// TIA Portal V16 export
// export: Created 2022-11-01T21:54:10.5360386Z, ExportSetting WithDefaults, DisplayName Totally Integrated Automation Portal, DisplayVersion V16, DisplayName TIA Portal Version Control Interface, DisplayVersion V16, DisplayName TIA Portal Openness, DisplayVersion V16, DisplayName SINAMICS Startdrive Advanced, DisplayVersion V16, DisplayName SINAMICS Startdrive G130, G150, S120, S150, SINAMICS MV, S210, DisplayVersion V16, DisplayName SINAMICS Startdrive G110M, G120, G120C, G120D, G120P, DisplayVersion V16, DisplayName STEP 7 Professional, DisplayVersion V16, DisplayName STEP 7 Safety, DisplayVersion V16, DisplayName WinCC Professional, DisplayVersion V16
VAR_GLOBAL   // PLC tag table "DI/O C900"
   iH120_Run_Km AT %M2900.0 : Bool;
   iH120_Con_Vfd AT %M2900.1 : Bool;
   iH120_Run_Vfd AT %M2900.2 : Bool;
   "qH120_Sel_Loc/Rem" AT %M2900.3 : Bool;
   "qH120_Sel_Km/Vfd" AT %M2900.4 : Bool;
   qH120_Block AT %M2900.5 : Bool;
   qH120_Connect_Vfd AT %M2900.6 : Bool;
   qH120_Start AT %M2900.7 : Bool;
   "iH615/1_Run_Km" AT %M2901.0 : Bool;
   "iH615/1_Con_Vfd" AT %M2901.1 : Bool;
   "iH615/1_Run_Vfd" AT %M2901.2 : Bool;
   "qH615/1_Sel_Loc/Rem" AT %M2901.3 : Bool;
   "qH615/1_Sel_Km/Vfd" AT %M2901.4 : Bool;
   "qH615/1_Block" AT %M2901.5 : Bool;
   "qH615/1_Connect_Vfd" AT %M2901.6 : Bool;
   "qH615/1_Start" AT %M2901.7 : Bool;
   "iH615/2_Run_Km" AT %M2902.0 : Bool;
   "iH615/2_Con_Vfd" AT %M2902.1 : Bool;
   "iH615/2_Run_Vfd" AT %M2902.2 : Bool;
   "qH615/2_Sel_Loc/Rem" AT %M2902.3 : Bool;
   "qH615/2_Sel_Km/Vfd" AT %M2902.4 : Bool;
   "qH615/2_Block" AT %M2902.5 : Bool;
   "qH615/2_Connect_Vfd" AT %M2902.6 : Bool;
   "qH615/2_Start" AT %M2902.7 : Bool;
   "iH616-x/1_Run_Km" AT %M2903.0 : Bool;
   "iH616-x/1_Con_Vfd" AT %M2903.1 : Bool;
   "iH616-x/1_Run_Vfd" AT %M2903.2 : Bool;
   "qH616-x/1_Sel_Loc/Rem" AT %M2903.3 : Bool;
   "qH616-x/1_Sel_Km/Vfd" AT %M2903.4 : Bool;
   "qH616-x/1_Block" AT %M2903.5 : Bool;
   "qH616-x/1_Connect_Vfd" AT %M2903.6 : Bool;
   "qH616-x/1_Start" AT %M2903.7 : Bool;
   "iH616-x/2_Run_Km" AT %M2904.0 : Bool;
   "iH616-x/2_Con_Vfd" AT %M2904.1 : Bool;
   "iH616-x/2_Run_Vfd" AT %M2904.2 : Bool;
   "qH616-x/2_Sel_Loc/Rem" AT %M2904.3 : Bool;
   "qH616-x/2_Sel_Km/Vfd" AT %M2904.4 : Bool;
   "qH616-x/2_Block" AT %M2904.5 : Bool;
   "qH616-x/2_Connect_Vfd" AT %M2904.6 : Bool;
   "qH616-x/2_Start" AT %M2904.7 : Bool;
   "iH900/1_Run_Km" AT %M2905.0 : Bool;
   "iH900/1_Con_Vfd" AT %M2905.1 : Bool;
   "iH900/1_Run_Vfd" AT %M2905.2 : Bool;
   "qH900/1_Sel_Loc/Rem" AT %M2905.3 : Bool;
   "qH900/1_Sel_Km/Vfd" AT %M2905.4 : Bool;
   "qH900/1_Block" AT %M2905.5 : Bool;
   "qH900/1_Connect_Vfd" AT %M2905.6 : Bool;
   "qH900/1_Start" AT %M2905.7 : Bool;
   "iH900/2_Run_Km" AT %M2906.0 : Bool;
   "iH900/2_Con_Vfd" AT %M2906.1 : Bool;
   "iH900/2_Run_Vfd" AT %M2906.2 : Bool;
   "qH900/2_Sel_Loc/Rem" AT %M2906.3 : Bool;
   "qH900/2_Sel_Km/Vfd" AT %M2906.4 : Bool;
   "qH900/2_Block" AT %M2906.5 : Bool;
   "qH900/2_Connect_Vfd" AT %M2906.6 : Bool;
   "qH900/2_Start" AT %M2906.7 : Bool;
   "iH901/1_Run_Km" AT %M2907.0 : Bool;
   "iH901/1_Con_Vfd" AT %M2907.1 : Bool;
   "iH901/1_Run_Vfd" AT %M2907.2 : Bool;
   "qH901/1_Sel_Loc/Rem" AT %M2907.3 : Bool;
   "qH901/1_Sel_Km/Vfd" AT %M2907.4 : Bool;
   "qH901/1_Block" AT %M2907.5 : Bool;
   "qH901/1_Connect_Vfd" AT %M2907.6 : Bool;
   "qH901/1_Start" AT %M2907.7 : Bool;
   "iH901/2_Run_Km" AT %M2908.0 : Bool;
   "iH901/2_Con_Vfd" AT %M2908.1 : Bool;
   "iH901/2_Run_Vfd" AT %M2908.2 : Bool;
   "qH901/2_Sel_Loc/Rem" AT %M2908.3 : Bool;
   "qH901/2_Sel_Km/Vfd" AT %M2908.4 : Bool;
   "qH901/2_Block" AT %M2908.5 : Bool;
   "qH901/2_Connect_Vfd" AT %M2908.6 : Bool;
   "qH901/2_Start" AT %M2908.7 : Bool;
   "iH902/1_Run_Km" AT %M2909.0 : Bool;
   "iH902/1_Con_Vfd" AT %M2909.1 : Bool;
   "iH902/1_Run_Vfd" AT %M2909.2 : Bool;
   "qH902/1_Sel_Loc/Rem" AT %M2909.3 : Bool;
   "qH902/1_Sel_Km/Vfd" AT %M2909.4 : Bool;
   "qH902/1_Block" AT %M2909.5 : Bool;
   "qH902/1_Connect_Vfd" AT %M2909.6 : Bool;
   "qH902/1_Start" AT %M2909.7 : Bool;
   "iH902/2_Run_Km" AT %M2910.0 : Bool;
   "iH902/2_Con_Vfd" AT %M2910.1 : Bool;
   "iH902/2_Run_Vfd" AT %M2910.2 : Bool;
   "qH902/2_Sel_Loc/Rem" AT %M2910.3 : Bool;
   "qH902/2_Sel_Km/Vfd" AT %M2910.4 : Bool;
   "qH902/2_Block" AT %M2910.5 : Bool;
   "qH902/2_Connect_Vfd" AT %M2910.6 : Bool;
   "qH902/2_Start" AT %M2910.7 : Bool;
   "iH904/1_Run_Km" AT %M2911.0 : Bool;
   "iH904/1_Con_Vfd" AT %M2911.1 : Bool;
   "iH904/1_Run_Vfd" AT %M2911.2 : Bool;
   "qH904/1_Sel_Loc/Rem" AT %M2911.3 : Bool;
   "qH904/1_Sel_Km/Vfd" AT %M2911.4 : Bool;
   "qH904/1_Block" AT %M2911.5 : Bool;
   "qH904/1_Connect_Vfd" AT %M2911.6 : Bool;
   "qH904/1_Start" AT %M2911.7 : Bool;
   "iH904/2_Run_Km" AT %M2912.0 : Bool;
   "iH904/2_Con_Vfd" AT %M2912.1 : Bool;
   "iH904/2_Run_Vfd" AT %M2912.2 : Bool;
   "qH904/2_Sel_Loc/Rem" AT %M2912.3 : Bool;
   "qH904/2_Sel_Km/Vfd" AT %M2912.4 : Bool;
   "qH904/2_Block" AT %M2912.5 : Bool;
   "qH904/2_Connect_Vfd" AT %M2912.6 : Bool;
   "qH904/2_Start" AT %M2912.7 : Bool;
   "iH905/1_Run_Km" AT %M2913.0 : Bool;
   "iH905/1_Con_Vfd" AT %M2913.1 : Bool;
   "iH905/1_Run_Vfd" AT %M2913.2 : Bool;
   "qH905/1_Sel_Loc/Rem" AT %M2913.3 : Bool;
   "qH905/1_Sel_Km/Vfd" AT %M2913.4 : Bool;
   "qH905/1_Block" AT %M2913.5 : Bool;
   "qH905/1_Connect_Vfd" AT %M2913.6 : Bool;
   "qH905/1_Start" AT %M2913.7 : Bool;
   "iH905/2_Run_Km" AT %M2914.0 : Bool;
   "iH905/2_Con_Vfd" AT %M2914.1 : Bool;
   "iH905/2_Run_Vfd" AT %M2914.2 : Bool;
   "qH905/2_Sel_Loc/Rem" AT %M2914.3 : Bool;
   "qH905/2_Sel_Km/Vfd" AT %M2914.4 : Bool;
   "qH905/2_Block" AT %M2914.5 : Bool;
   "qH905/2_Connect_Vfd" AT %M2914.6 : Bool;
   "qH905/2_Start" AT %M2914.7 : Bool;
   "iD601/1_Run_Km" AT %M2915.0 : Bool;
   "iD601/1_Con_Vfd" AT %M2915.1 : Bool;
   "iD601/1_Run_Vfd" AT %M2915.2 : Bool;
   "qD601/1_Sel_Loc/Rem" AT %M2915.3 : Bool;
   "qD601/1_Sel_Km/Vfd" AT %M2915.4 : Bool;
   "qD601/1_Block" AT %M2915.5 : Bool;
   "qD601/1_Connect_Vfd" AT %M2915.6 : Bool;
   "qD601/1_Start" AT %M2915.7 : Bool;
   "iD601/2_Run_Km" AT %M2916.0 : Bool;
   "iD601/2_Con_Vfd" AT %M2916.1 : Bool;
   "iD601/2_Run_Vfd" AT %M2916.2 : Bool;
   "qD601/2_Sel_Loc/Rem" AT %M2916.3 : Bool;
   "qD601/2_Sel_Km/Vfd" AT %M2916.4 : Bool;
   "qD601/2_Block" AT %M2916.5 : Bool;
   "qD601/2_Connect_Vfd" AT %M2916.6 : Bool;
   "qD601/2_Start" AT %M2916.7 : Bool;
   "iD901/1_Run_Km" AT %M2917.0 : Bool;
   "iD901/1_Con_Vfd" AT %M2917.1 : Bool;
   "iD901/1_Run_Vfd" AT %M2917.2 : Bool;
   "qD901/1_Sel_Loc/Rem" AT %M2917.3 : Bool;
   "qD901/1_Sel_Km/Vfd" AT %M2917.4 : Bool;
   "qD901/1_Block" AT %M2917.5 : Bool;
   "qD901/1_Connect_Vfd" AT %M2917.6 : Bool;
   "qD901/1_Start" AT %M2917.7 : Bool;
   "iD901/2_Run_Km" AT %M2918.0 : Bool;
   "iD901/2_Con_Vfd" AT %M2918.1 : Bool;
   "iD901/2_Run_Vfd" AT %M2918.2 : Bool;
   "qD901/2_Sel_Loc/Rem" AT %M2918.3 : Bool;
   "qD901/2_Sel_Km/Vfd" AT %M2918.4 : Bool;
   "qD901/2_Block" AT %M2918.5 : Bool;
   "qD901/2_Connect_Vfd" AT %M2918.6 : Bool;
   "qD901/2_Start" AT %M2918.7 : Bool;
   "iD902/1_Run_Km" AT %M2919.0 : Bool;
   "iD902/1_Con_Vfd" AT %M2919.1 : Bool;
   "iD902/1_Run_Vfd" AT %M2919.2 : Bool;
   "qD902/1_Sel_Loc/Rem" AT %M2919.3 : Bool;
   "qD902/1_Sel_Km/Vfd" AT %M2919.4 : Bool;
   "qD902/1_Block" AT %M2919.5 : Bool;
   "qD902/1_Connect_Vfd" AT %M2919.6 : Bool;
   "qD902/1_Start" AT %M2919.7 : Bool;
   "iD902/2_Run_Km" AT %M2920.0 : Bool;
   "iD902/2_Con_Vfd" AT %M2920.1 : Bool;
   "iD902/2_Run_Vfd" AT %M2920.2 : Bool;
   "qD902/2_Sel_Loc/Rem" AT %M2920.3 : Bool;
   "qD902/2_Sel_Km/Vfd" AT %M2920.4 : Bool;
   "qD902/2_Block" AT %M2920.5 : Bool;
   "qD902/2_Connect_Vfd" AT %M2920.6 : Bool;
   "qD902/2_Start" AT %M2920.7 : Bool;
   iH906_Run_Km AT %M2921.0 : Bool;
   iH906_Con_Vfd AT %M2921.1 : Bool;
   iH906_Run_Vfd AT %M2921.2 : Bool;
   "qH906_Sel_Loc/Rem" AT %M2921.3 : Bool;
   "qH906_Sel_Km/Vfd" AT %M2921.4 : Bool;
   qH906_Block AT %M2921.5 : Bool;
   qH906_Connect_Vfd AT %M2921.6 : Bool;
   qH906_Start AT %M2921.7 : Bool;
END_VAR
